FUNCTION_BLOCK StartAfterNoConfig (* Basic Function Block Type *)
  (* Standard: 61499-2 *)
  (* Version 0.0, 7/11/2026, Schneider Electric, Template *)
  PACKAGE SE.Nereda;
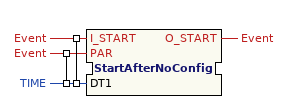
  EVENT_INPUT
    I_START WITH DT1;
    PAR WITH DT1;
  END_EVENT
  EVENT_OUTPUT
    O_START;
  END_EVENT
  VAR_INPUT
    DT1 : TIME;
  END_VAR
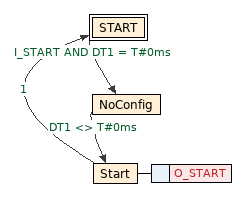
  EC_STATES
    START; (* Initial State *)
    NoConfig;
    Start : -> O_START;
  END_STATES
  EC_TRANSITIONS
    START TO NoConfig := I_START AND DT1 = T#0ms;
    NoConfig TO Start := DT1 <> T#0ms;
    Start TO START := 1;
  END_TRANSITIONS
  ALGORITHM INIT IN ST: (* Initialization algorithm *)
;
  END_ALGORITHM
  ALGORITHM REQ IN ST: (* Normally executed algorithm *)
;
  END_ALGORITHM
END_FUNCTION_BLOCK
